Fanuc KAREL source: NC0004.KL

-- PROVISIONAL review KL for V940-1; original PC SHA256 4089c896c9cf8f99abdb14dcb8a92c608f1adf2b50850793507aaa1964d2034c
-- Incomplete behavior may be omitted. Consult companion uncertainty JSON. Do not deploy.
PROGRAM NC0004
%NOLOCKGROUP
-- UNRESOLVED_LOCAL_POOL 1 cells at code offset 3; source declarations unknown
-- DIRECT_LOCAL_WORD_ACCESS alone does not prove INTEGER, REAL, or BOOLEAN
BEGIN
  -- V9_EXPOSED_INDEXED_TABLE_HINT layout=0001; 6 counted words exposed once; source arms/runtime held
  -- V9_CONDITION_STACK_HINT 3 bounded expression windows; static native code-base-relative target link; source arms held
  -- UNRESOLVED_PC offsets 0-8; opcodes 2B,2C,7B
  -- UNRESOLVED_PC offsets 13-20; opcodes 9D,23
  -- UNRESOLVED_PC offsets 25-38; opcodes 21,9D,57,79
  -- UNRESOLVED_PC offsets 43-56; opcodes 21,9D,57,79
  -- UNRESOLVED_PC offsets 61-74; opcodes 21,9D,57,79
  -- UNRESOLVED_PC offsets 79-93; opcodes 21,9D,52,23
  -- UNRESOLVED_PC offsets 98-103; opcodes 7A
  -- UNRESOLVED_PC offsets 108-126; opcodes 21,2E,52,23
  -- UNRESOLVED_PC offsets 136-141; opcodes 7A
  -- UNRESOLVED_PC offsets 146-164; opcodes 21,2E,52,23
  -- UNRESOLVED_PC offsets 174-179; opcodes 7A
  -- UNRESOLVED_PC offsets 184-202; opcodes 21,2E,52,23
  -- UNRESOLVED_PC offsets 212-216; opcodes 7F
  -- UNRESOLVED_PC offsets 221-225; opcodes 27,AA
  -- UNRESOLVED_PC offsets 230-234; opcodes 7F
END NC0004
